// TIA Portal V20 export
DATA_BLOCK "SYSTEM_DB"   // DB1990
{ S7_Optimized_Access := 'TRUE' }
AUTHOR : Tesla
FAMILY : Base
VERSION : 1.0
// stored: MemoryReserve 0
   VAR
      Init_HMI_OPmode { ExternalAccessible := 'False'; ExternalVisible := 'False'; ExternalWritable := 'False'; S7_SetPoint := 'True'} : "INIT_HMI_OPMODE_UDT";   // Initial Werte / HMI操作模式初始化 / Init 值
      OPmode { S7_SetPoint := 'True'} : Array[0.."No_OperationMODE"] of "OPMODE_UDT";   // Operation mode / 操作模式 / 运行 模式
      HMI_Panel { ExternalAccessible := 'False'; ExternalVisible := 'False'; ExternalWritable := 'False'; S7_SetPoint := 'True'} : Array[0.."No_HMI_PANEL"] of "HMI_PANEL_UDT";   // HMI / Panel
      HMI_GLOBAL { ExternalAccessible := 'False'; ExternalVisible := 'False'; ExternalWritable := 'False'; S7_SetPoint := 'True'} : "GLOBAL_STRUCT_UDT";
   END_VAR
BEGIN
   // Init_HMI_OPmode.OPmode_init : 操作模式初始化值
   // Init_HMI_OPmode.HMI_Panel_init : HMI 操作面板初始化值
   // Init_HMI_OPmode.OPmode_activated : 操作模式激活信息
   // Init_HMI_OPmode.HMI_Panel_No : 分配面板到操作模式区域
END_DATA_BLOCK
